{attribute 'enable_dynamic_creation'}
FUNCTION_BLOCK Notification IMPLEMENTS Object
VAR
	sNotification : STRING;
END_VAR

METHOD FB_init : BOOL
VAR_INPUT
	bInitRetains : BOOL; // if TRUE, the retain variables are initialized (warm start / cold start)
	bInCopyCode : BOOL;  // if TRUE, the instance afterwards gets moved into the copy code (online change)
	sNotification : STRING;
END_VAR
THIS^.sNotification := sNotification;
END_METHOD

METHOD getNotification : STRING
VAR_INPUT
END_VAR
getNotification := THIS^.sNotification;
END_METHOD

END_FUNCTION_BLOCK

(* stored: Version 1.1.0.1, ProductVersion 3.1.4024.12
   POU Notification: Id {eed2ee3d-6fd1-4636-bf5e-23c81a254f4a}, SpecialFunc None
   Method FB_init: Id {ccd27d29-8515-4b75-9379-b5f629f9d933}
   Method getNotification: Id {fa7571e4-c8c8-4de4-8b52-f7469a8bf617} *)
